// SIMATIC STEP 7 (V5.x) project EuroAsiaFood_V00_00_01
// CPU: CPU 314C-2 PN/DP
// station: Hardware
// station: SIMATIC 300(1)
// station: P_ADR_BUS
// program: S7-Programm(1)

SYMBOL_TABLE
"DB1 Weight Logging"	DB 1	FB 1	// Wiegemitschreibung
"DB2 Simulation"	DB 2	FB 2	// Simulation der Anlage
"DB3 global Info"	DB 3	DB 3	// globale Programm- / Fehlerinformationen
"DB4 Motor Data for FCs"	DB 4	DB 4	// Motordaten für Frequenzumformer
"DB5 reserve"	DB 5	DB 5	// reserve
"DB6 reserve"	DB 6	DB 6	// reserve
"DB7 SiSc-Par WS-Communic"	DB 7	DB 7	// Lagerort-Waagenparameter für WS Kopplung
"DB8 Batch Info from PC"	DB 8	DB 8	// Chargeninfo von PC
"DB9 reserve"	DB 9	DB 9
"DB10 Scale Configuration"	DB 10	DB 10	// Waagenkonfiguration
"DB11 Com DB Recipe Data"	DB 11	DB 11	// Koppel-DB Rezeptdaten
"DB12 Com-DB S-S Param"	DB 12	DB 12	// Koppel-DB Silo-Waagen-Parameter
"DB13 Scale Par from PC"	DB 13	DB 13	// SST Waagenparameter von PC
"DB14 Scale Par to PC"	DB 14	DB 14	// SST Waagenparameter zu PC
"DB15 R->C Level scale(S)"	DB 15	DB 15	// SST Rezeptebene -> Komponentenebene Waage Steuer-/Status
"DB16 R->C Level(D)"	DB 16	DB 16	// Interface recipe level  -> component level scale Data
"DB17 C->R Level Scale"	DB 17	DB 17	// SST Komponentneebene -> Rezeptebene Waage
"DB18 R<->C-Level Scale(A"	DB 18	DB 18	// SST Komponentneebene <-> Rezeptebene Waage Zusatzdaten
"DB19 DB Act Scale Data"	DB 19	DB 19	// Waagenistdaten-DB
"DB20 IF SC1 Control-DB"	DB 20	FB 15	// SST FG 1 <-> SPS-Waage Steuer-DB
"DB21 IF SC1 Scale Par"	DB 21	DB 21	// SST FG 1 <-> SPS-Waage Waagenparameter
"DB22 IF SC1 Recipe Data"	DB 22	DB 22	// SST FG 1 <-> SPS-Waage Lagerort-/Rezeptdaten
"DB23 IF SC2 Control-DB"	DB 23	FB 15	// SST FG 2 <-> SPS-Waage Steuer-DB
"DB24 IF SC2 Scale Par"	DB 24	DB 24	// SST FG 2 <-> SPS-Waage Waagenparameter
"DB25 IF SC2 Recipe Data"	DB 25	DB 25	// SST FG 2 <-> SPS-Waage Lagerort-/Rezeptdaten
"DB26 IF SC3 Control-DB"	DB 26	FB 15	// SST FG 3 <-> SPS-Waage Steuer-DB
"DB27 IF SC3 Scalen Par"	DB 27	DB 27	// SST FG 3 <-> SPS-Waage Waagenparameter
"DB28 IF SC3 Recipe Data"	DB 28	DB 28	// SST FG 3 <-> SPS-Waage Lagerort-/Rezeptdaten
"DB29 reserve"	DB 29	DB 29	// reserve
"DB30 Daten from/to SCADA"	DB 30	FB 30
"DB31 Mode to SCADA"	DB 31	DB 31	// Betriebsmode der Objekte zu Farbgrafik
"DB32 Inputs"	DB 32	FB 32
"DV33 Outputs"	DB 33	FB 33
"DB34 Faults"	DB 34	FB 34	// Anlagenstörungen
"DB35 Acknowledge Faults"	DB 35	DB 35	// Quittierungen
"DB36 Operating notific"	DB 36	DB 36	// Betriebsmeldungen
"DB37Service warning msg"	DB 37	DB 37	// Service Warnmeldungen
"DB38 Service fault msg"	DB 38	DB 38	// Service Störmeldungen
"DB39 free Data for SCADA"	DB 39	DB 39	// freie Datenaufzeichnung über Visualisierung
"DB40 IF SC4 Control-DB"	DB 40	FB 15	// SST FG 4 <-> SPS-Waage Steuer-DB
"DB41 IF SC4 Scale Par"	DB 41	DB 41	// SST FG 4 <-> SPS-Waage Waagenparameter
"DB42 IF SC4 Recipe Data"	DB 42	DB 42	// SST FG 4 <-> SPS-Waage Lagerort-/Rezeptdaten
"DB43 IF SC5 Control-DB"	DB 43	FB 15	// SST FG 5 <-> SPS-Waage Steuer-DB
"DB44 IF SC5 Scale Par"	DB 44	DB 44	// SST FG 5 <-> SPS-Waage Waagenparameter
"DB45 IF SC5 Recipe Data"	DB 45	DB 45	// SST FG 5 <-> SPS-Waage Lagerort-/Rezeptdaten
"DB46 IF SC6 Control-DB"	DB 46	FB 15	// SST FG 6 <-> SPS-Waage Steuer-DB
"DB47 IF SC6 Scale Par"	DB 47	DB 47	// SST FG 6 <-> SPS-Waage Waagenparameter
"DB48 IF SC6 Recipe Data"	DB 48	DB 48	// SST FG 6 <-> SPS-Waage Lagerort-/Rezeptdaten
"DB49 reserve"	DB 49	DB 49	// reserve
"DB50 Control bits PC"	DB 50	DB 50	// Steuerbitleiste von/zu PC
"DB51 Manual Addition PC"	DB 51	DB 51	// Quittierung Handzugaben / Daten Handzugaben von/zu PC
"DB52 Batch Info PC"	DB 52	DB 52	// Chargeninformationen von PC (Rezeptnr./Chargennr. usw.)
"DB53 Consumer Info PC"	DB 53	DB 53	// Verbraucherinformationen von/zu PC
"DB54 Transponder Info PC"	DB 54	DB 54	// Transponderinfprmationen von/zu PC
"DB55 Silo Info PC"	DB 55	DB 55	// Siloinformationen von/zu PC
"DB56 Silo Refill"	DB 56	DB 56	// Silonachfüllung von/zu PC
"DB57 List Man Addition"	DB 57	DB 57	// Handzugabeliste zur Anzeige auf OP oder FG)
"DB58 Project spec. res."	DB 58	DB 58	// reserve
"DB59 Mixer Values"	DB 59	DB 59	// Mischerwerte an PC
"DB60 Mixer Step Info"	DB 60	DB 60	// Mischerschrittinformationen an PC
"DB61 Mix Recipe M1"	DB 61	DB 61	// Mixer Recipe Mixerer 1 bzw. Heating Mixer 1 and Cooling Mixerer 1 from PC
"DB62 Mix Recipe M2"	DB 62	DB 62	// Mixer recipe mixer 2 or heater mixer 2 and cooler mixer 2 from PC
"DB63 Mix Recipe M3"	DB 63	DB 63	// Mixer recipe mixer 3 or heater mixer 3 and cooler mixer 3 from PC
"DB64 Mix Recipe M4"	DB 64	DB 64	// Mixer recipe mixer 4 or heater mixer 4 and cooler mixer 4 from PC
"DB65 Mix Recipe M5"	DB 65	DB 65	// Mixer recipe mixer 5 or heater mixer 5 and cooler mixer 5 from PC
"DB66 Mix Recipe M6"	DB 66	DB 66	// Mixer recipe mixer 6 or heater mixer 6 and cooler mixer 6 from PC
"DB67 Mix Recipe M7"	DB 67	DB 67	// Mixer recipe mixer 7 or heater mixer 7 and cooler mixer 7 from PC
"DB68 Mix Recipe M8"	DB 68	DB 68	// Mixer recipe mixer 8 or heater mixer 8 and cooler mixer 8 from PC
"DB69 Mix Recipe M9"	DB 69	DB 69	// Mixer recipe mixer 9 or heater mixer 9 and cooler mixer 9 from PC
"DB70 IF OP1 Control-DB"	DB 70	FB 16	// SST OP 1 <-> SPS-Waage Steuer-DB
"DB71 IF OP1 Scale Par"	DB 71	DB 71	// SST OP 1 <-> SPS-Waage Waagenparameter
"DB72 IF OP1 Recipe Datan"	DB 72	DB 72	// SST OP 1 <-> SPS-Waage Lagerort-/Rezeptdaten
"DB73 IF OP2 Control-DB"	DB 73	FB 16	// SST OP 2 <-> SPS-Waage Steuer-DB
"DB74 IF OP2 Scale Par"	DB 74	DB 74	// SST OP 2 <-> SPS-Waage Waagenparameter
"DB75 IF OP2 Recipe Data"	DB 75	DB 75	// SST OP 2 <-> SPS-Waage Lagerort-/Rezeptdaten
"DB90 Shuttle-DB"	DB 90	DB 90	// Shuttle-DB
"DB91 ContainerDB Shuttle"	DB 91	DB 91	// Container-DB Shuttle
"DB92 Station-DB Shuttle"	DB 92	DB 92	// Stations-DB Shuttle
"PRODUCTION_DB"	DB 1000	FB 1000	// Call Line 1 DB
"HOPPER_HP01_DB"	DB 1001	FB 1001
"HOPPER_HP02_DB"	DB 1002	FB 1001
"REC01_DB"	DB 1011	FB 1011	// Receiver REC01
"PMP01_DB"	DB 1051	FB 1051
"FC01_RV_HOPPERS_DB"	DB 10001	FB 4901
"Example DB read table"	DB 60000	DB 60000	// Beispiel-DB Tabelle auslesen
"R->C Level Scale (S)"	DB 60201	DB 60201	// SST Rezeptebene -> Komponentenebene Waage Steuer-/Status
"R->C Level Scale (D)"	DB 60202	DB 60202	// SST Rezeptebene -> Komponentenebene Waage Daten
"K->S Level Scale (S)"	DB 60203	DB 60203	// SST Komponentenebene -> Einzelschrittebene Waage Steuer-/Status
"K->S Level Scale (D)"	DB 60204	DB 60204	// Interface component level -> single step level Scale Daten
"S->A Level Scale (S)"	DB 60205	DB 60205	// SST Einzelschrittebene -> Analogebene Waage Steuer-/Status
"S->A Level Scale (D)"	DB 60206	DB 60206	// SST Einzelschrittebene -> Analogebene Waage Daten
"K->R Level Scale"	DB 60207	DB 60207	// SST Komponentneebene -> Rezeptebene Waage
"S->C Level Scale"	DB 60208	DB 60208	// SST Einzelschrittebene -> Komponentenebene Waage
"A->S Level Scale"	DB 60209	DB 60209	// SST Analogebene -> Einzelschrittebene Waage
"IF SCADA Control-DB"	DB 60211	DB 60211	// Schnittstelle zu Farbgrafik Steuer-DB
"IF SCADA Scale Par"	DB 60212	DB 60212	// Schnittstelle zu Farbgrafik Waagenparameter
"IF SCADA RecipeData"	DB 60213	DB 60213	// Schnittstelle zu Farbgrafik Rezeptdaten
"IF SCADA 1 Control-DB"	DB 60250	DB 60250	// SST FG 1 <-> SPS-Waage Steuer-DB
"Mixer Recipe-DB"	DB 60300	DB 60300	// Mixer recipe DB
"FB1 Weight logging"	FB 1	FB 1	// Wiegemitschreibung
"FB2 Simulation"	FB 2	FB 2	// Simulation der Anlage
"FB3 Mix Recipe Interpr."	FB 3	FB 3	// Mischrezeptinterpreter
"FB4 Freq Converter L2"	FB 4	FB 4	// Frequenzumformer L2-Bus
"FB5 Componenter_L2"	FB 5	FB 5	// Componenter L2-Bus
"FB6 reserve"	FB 6	FB 6	// reserve
"FB7 Rot Diverter Valve"	FB 7	FB 7	// Saugrohrverteiler
"FB8 reserve"	FB 8	FB 8	// reserve
"FB9 Pos. Pipe Diverter"	FB 9	FB 9	// Wegstellung (Rohrweiche)
"FB10 Order Level"	FB 10	FB 10	// Auftragsebene Waage
"FB11 Recipe Level"	FB 11	FB 11	// Rezeptebene Waage
"FB12 Component Level"	FB 12	FB 12	// Komponentenebene Waage
"FB13 Single Step Level"	FB 13	FB 13	// Single step level scale
"FB14 Analogue Level"	FB 14	FB 14	// Analogue level scale
"FB15 IF PLC-Scale/SCADA"	FB 15	FB 15	// Schnittstelle SPS-Waage / Farbgrafik
"FB16 IF PLC-Scale/OP"	FB 16	FB 16	// Schnittstelle SPS-Waage / OP
"FB17 IF PLC-Scale/HSH"	FB 17	FB 17	// Schnittstelle SPS-Waage / HSH
"FB18 IF PLC-Scale/OP OL"	FB 18	FB 18	// Schnittstelle SPS-Waage / OP Auftragebene
"FB19 IF PLC-Scale/Bil"	FB 19	FB 19	// Schnittstelle SPS-Waage / Farbgrafik Bilanzen
"FB20 Siwarex-U Comm"	FB 20	FB 20	// SPS-Waage Siwarex-U Kopplung
"FB21 MCS-DMV Comm"	FB 21	FB 21	// SPS-Waage MCS-DMV Kopplung
"FB22 MV1 Comm"	FB 22	FB 22	// SPS-Waage MV1 Kopplung
"FB23 Siwarex-M Comm"	FB 23	FB 23	// SPS-Waage Siwarex-M Kopplung
"FB25 Promass 63 Comm"	FB 25	FB 25	// SPS-Waage Promass 63 Kopplung
"FB26 Pulse Count FM350-2"	FB 26	FB 26	// SPS-Waage Impulszähler FM350-2 Kopplung
"FB27 PESA"	FB 27	FB 27	// SPS-Waage PESA Modul Kopplung
"FB28 Bizerba"	FB 28	FB 28	// SPS-Waage Bizerba Modul Kopplung
"FB29 Mettler-Scale ID7"	FB 29	FB 29	// SPS-Waage Mettler-ID7
"FB30 Daten from/to SCADA"	FB 30	FB 30	// Daten von / an Farbgrafik
"FB31 Mode Obj. to SCADA"	FB 31	FB 31	// Mode Objekte an Farbgrafik OP
"FB32 Inputs to SCADA"	FB 32	FB 32	// Eingänge an Farbgrafik / OP
"FB33 Outputs to SCADA"	FB 33	FB 33	// Ausgänge an Farbgrafik / OP
"FB34 Fault evaluation"	FB 34	FB 34	// Störauswertung
"FB36 WMD ET200M"	FB 36	FB 36	// SPS-Waage WMD Kopplung
"FB37 Pulse Count FM350-1"	FB 37	FB 37	// PLC-scale Pulse Counter FM 350-1
"FB38 gwt PR5210"	FB 38	FB 38	// SPS-Waage gwt PR5210
"FB39 WMD Bürkert"	FB 39	FB 39	// SPS-Waage WMD Bürkert
"FB40 Weight Siware- U"	FB 40	FB 40	// Gewichtswert von Siwarex U
"FB41 Weight MCS-DMV"	FB 41	FB 41	// Gewichtswert von MCS-DMV
"FB42 Weight MV1"	FB 42	FB 42	// Gewichtswert von MV1
"FB43 Weight Siwarex-M"	FB 43	FB 43	// Gewichtswert von Siwarex M
"FB45 LiW  DISOCONT"	FB 45	FB 45	// Differentialdosierwaage DSIOCONT
"FB46 IF LiW / SCADA"	FB 46	FB 46	// Schnittstelle DISOCONT Differentialdosierwaage / Farbgrafik
"FB47 IF LiW / OP"	FB 47	FB 47	// Schnittstelle DISOCONT Differentialdosierwaage / OP
"FB50 Control signals PC"	FB 50	FB 50	// Steuerbits von/an PC
"FB51 Manual addition"	FB 51	FB 51	// Quittierung Handzugaben / Daten Handzugabe
"FB52 Batch Info"	FB 52	FB 52	// Chargeninformationen (Rezept Nr./Chargennummer usw.)
"FB53 Consumer Info"	FB 53	FB 53	// Verbraucherinformationen von/zu PC
"FB54 Transponder Info"	FB 54	FB 54	// Transponderinformationen von/zu PC
"FB55 Silo Info PC"	FB 55	FB 55	// Siloinformationen von/zu PC
"FB56 Silo Refill"	FB 56	FB 56	// Silonachfüllung von/zu PC
"FB71 Siwarex CS"	FB 71	FB 71	// SPS-Waage Siwarex CS Kopplung Analogebene
"FB72 Siwarex CS_DR"	FB 72	FB 72	// SPS-Waage Siwarex CS Kopplung Siemens "SICS_DR"
"FB73 Siwarex CS_BA"	FB 73	FB 73	// SPS-Waage Siwarex CS Kopplung Siemens "SICS_BA"
"FB74 Counter ET200S"	FB 74	FB 74	// SPS-Waage Impulszähler über ET200S 1Count 24V/100kHz
"FB75 Mettler Jaguar"	FB 75	FB 75	// SPS-Waage Mettler Jaguar
"FB76 Siwarex FTA"	FB 76	FB 76	// SPS-Waage Siwarex FTA
"FB77 FB Siwarex FTA"	FB 77	FB 77	// SPS-Waage FB Siwarex FTA Siemens Funktionsbaustein
"FB78 Mettler PB-Module"	FB 78	FB 78	// SPS-Waage Mettler Profibus-Modul
"FB79 Mettler IND690"	FB 79	FB 79	// SPS-Waage Mettler IND690
"FB80 DK800"	FB 80	FB 80	// SPS-Waage DK800
"FB81 Promag 50"	FB 81	FB 81	// SPS-Waage Promag 50
"FB82 Mettler Panther"	FB 82	FB 82	// SPS-Waage Mettler Panther
"FB90 Shuttle-FB"	FB 90	FB 90	// Shuttle-FB
"FB91 ContainerFB Shuttle"	FB 91	FB 91	// Container-FB Shuttle
"FB92 Stations-FB Shuttle"	FB 92	FB 92	// Stations-FB Shuttle
"PRODUCTION"	FB 1000	FB 1000	// Call Line FBs
"HOPPER"	FB 1001	FB 1001	// HP01 and HP02
"REC01"	FB 1011	FB 1011	// Receiver REC01
"PMP01"	FB 1051	FB 1051
"BLOWER_P01"	FB 1081	FB 1081	// Pressure Blower
"FC01_RV_HOPPERS"	FB 4901	FB 4901	// Frequncy Converter rotary valves HP01/HP02
"FC1 Cycle Gen Timer"	FC 1	FC 1	// Taktgeber mit Timervorgabe
"FC2 Cycle Gen Timer Emul"	FC 2	FC 2	// Taktgeber mit Timernachbildung
"FC3 Cycle generator"	FC 3	FC 3	// Timernachbildung SA,SE,SV,SI
"FC4 Block transfer ANY"	FC 4	FC 4	// Block transferieren mit ANY-Zeiger
"FC5 Block Transfer"	FC 5	FC 5	// Block transferieren, Datenwort schreiben
"FC6 Set/Query Data Bit"	FC 6	FC 6	// Datenbit zuweisen oder abfragen
"FC7 Read Table"	FC 7	FC 7	// Eintrag aus Tabelle auslesen
"FC8 Determin ANY-Pointer"	FC 8	FC 8	// ANY-Zeiger in DB,DW,Länge zerlegen
"FC9 Set path"	FC 9	FC 9	// Weg stellen (Rohrweichen)
"FC10 Analogue value r/w"	FC 10	FC 10	// Analogwert lesen/schreiben
"FC11 PressureTransmitter"	FC 11	FC 11	// Drucktransmitterwert einlesen
"FC12 Restart"	FC 12	FC 12	// Neu- / Wiedeanlauf
"FC13 Standard Signals"	FC 13	FC 13	// Standardsignale
"FC14 Debounce Indicator"	FC 14	FC 14	// Melder entprellen
"FC15 I/O-FAT/Simulation"	FC 15	FC 15	// E/A FAT / Simulation
"FC16 Fault evaluation"	FC 16	FC 16	// Störauswertung
"FC17 String compare"	FC 17	FC 17	// Stringvergleich
"FC18 FIFO/LIFO"	FC 18	FC 18	// FIFO/LIFO
"FC19 Motor 2O2I"	FC 19	FC 19	// Motor Objekt 2 (2 Ausgänge, 2 Eingänge)
"FC20 Motor 1O1I"	FC 20	FC 20	// Motor Objekt 1 (1 Ausgang, 1 Eingang)
"FC21 Valve 10-2I"	FC 21	FC 21	// Ventil Objekt 1 (1 Ausgang, 0-2 Eingänge)
"FC22 Valve 2O2I"	FC 22	FC 22	// Ventil Objekt 2 (2 Ausgänge, 2Eingänge)
"FC23 Valve 1-10O"	FC 23	FC 23	// Ventil Objekt 3 (Ansteuerung von max. 10 getakteten Ventilen)
"FC24 Binary-I Object"	FC 24	FC 24	// Binär-Eingangs Objekt
"FC25 Pipe Diverter 3O3I"	FC 25	FC 25	// Pipe Diverter 3 Outputs, 3 inputs
"FC26 DosingValve 2O2I"	FC 26	FC 26	// Dosierventil grob/fein 2 Ausgänge, 2 Eingänge)
"FC30 Pre -assign DB"	FC 30	FC 30	// Datenbaustein vorbelegen
"FC31 PLC-Scale"	FC 31	FC 31	// Aufruf SPS-Waage
"FC32 Rec/Comp r/w/d"	FC 32	FC 32	// Rezept/Komponente lesen/schreiben/löschen
"FC33 Si/Rec from PC r/w"	FC 33	FC 33	// Lagerortparameter von PC lesen/schreiben
"FC34 Si/Sc Par r/w"	FC 34	FC 34	// Silo-/Waagenparameter lesen/schreiben
"FC35 reserve Scale"	FC 35	FC 35
"FC36 Si-Configuration"	FC 36	FC 36	// Lagerortkonfiguration
"FC37 Si/Sc Par r/w"	FC 37	FC 37	// Lagerortparameter einer Siwarex-Waage lesen/schreiben
"FC38 reserve Scale"	FC 38	FC 38
"FC39 Siwarex-M"	FC 39	FC 39	// Kommunikationsbaustein Siwarex-M
"FC40 copy Obj-IF Master"	FC 40	FC 40	// Objekt-Schnittstelle kopieren Master
"FC41 copy Obj-IF Slave"	FC 41	FC 41	// Objekt-Schnittstelle kopieren Slave
"FC43 FM350-2"	FC 43	FC 43
"FC44 FM350-2 I/O"	FC 44	FC 44
"FC45 Data Promass 63"	FC 45	FC 45	// Daten von Promass 63 DP
"FC47 Write Table"	FC 47	FC 47	// Eintrag in Tabelle schreiben
"FC50 LiW Scale DISOCONT"	FC 50	FC 50	// FC50 Aufruf DISOCONT Differentialdosierwaage
"FC60 Silo Pilot"	FC 60	FC 60	// Silopilot
"FC61 Bürkert DosingValve"	FC 61	FC 61	// Bürkert Dosierventil
"FC62 Analogue Valve"	FC 62	FC 62	// Analogventil
"FC64 aux fct registr"	FC 64	FC 64	// Hilfsfunktion Registrierung
"FC65 scale-db-no"	FC 65	FC 65
"FC66 info functiontime"	FC 66	FC 66
"EUi_02_04_201"	I 4.0	BOOL	// production area PMP01 motor vacuum pump
"EUi_02_01_201"	I 4.1	BOOL	// production area REC01 motor rotary valev
"EUi_02_02_201"	I 4.2	BOOL	// production area SM01 motor screener
"EUi_02_02_202"	I 4.3	BOOL	// production area SM01 motor magnetic seperator
"EUi_01_01_201"	I 4.4	BOOL	// material preparation HP01 motor rotary valve
"EUi_01_02_201"	I 4.5	BOOL	// material preparation HP02 motor rotary valve
"Ln_01_01_301"	I 4.6	BOOL	// material preparation HP01 low level sensor indicator
"Ln_01_02_301"	I 4.7	BOOL	// material preparation HP01 low level sensor indicator
"HZ_02_04_201"	I 5.0	BOOL	// production area PMP01 motor vacuum pump
"HZ_02_01_201"	I 5.1	BOOL	// production area REC01 motor rotary valve
"HZ_02_02_201"	I 5.2	BOOL	// production area SM01 motor screener
"HZ_02_02_202"	I 5.3	BOOL	// production area SM01 motor magnetic seperator
"HZ_01_01_201"	I 5.4	BOOL	// material preparation HP01 motor rotary valve
"HZ_01_02_201"	I 5.5	BOOL	// material preparation HP02 motor rotary valve
"ES_03_01_601"	I 5.6	BOOL	// system system input emergency stop ok
"ES_03_01_602"	I 5.7	BOOL	// system system input fault fuse
"GZ_02_01_601"	I 6.0	BOOL	// production area REC01 input safety circuit
"GZ_02_02_601"	I 6.1	BOOL	// production area SM01 input safety circuit
"GZ_01_01_601"	I 6.2	BOOL	// material preparation HP01 input safety circuit
"GZ_01_02_601"	I 6.3	BOOL	// material preparation HP02 input safety circuit
"Gn_02_01_602"	I 6.4	BOOL	// production area REC01 input rotor monitoring
"Gn_01_01_602"	I 6.5	BOOL	// material preparation HP01 input rotor monitoring
"Gn_01_02_602"	I 6.6	BOOL	// material preparation HP02 input rotor monitoring
"I 6.7"	I 6.7	BOOL	// free
"Lp_02_01_301"	I 10.0	BOOL	// production area REC01 sensor high level indicator
"Ln_02_01_302"	I 10.1	BOOL	// production area REC01 sensor low level indicator
"Lp_02_03_301"	I 10.2	BOOL	// production area HP03 sensor high level indicator
"Ln_02_03_302"	I 10.3	BOOL	// production area HP03 sensor low level indicator
"Gp_01_02_102"	I 10.4	BOOL	// material preparation HP02 valve outlet flap
"EUi_01_01_202"	I 10.5	BOOL	// material preparation HP01 motor vibrator
"EUi_01_02_202"	I 10.6	BOOL	// material preparation HP02 motor vibrator 1
"EUi_01_02_203"	I 10.7	BOOL	// material preparation HP02 motor vibrator 2
"HZ_01_01_202"	I 11.0	BOOL	// material preparation HP01 motor vibrator
"HZ_01_02_202"	I 11.1	BOOL	// material preparation HP02 motor vibrator 1
"HZ_01_02_203"	I 11.2	BOOL	// material preparation HP02 motor vibrator 2
"ES_02_03_601"	I 11.3	BOOL	// production area HP03 input PFC ready
"ES_02_03_602"	I 11.4	BOOL	// production area HP03 input PFC take material
"ES_01_02_603"	I 11.5	BOOL	// production area HP03 input PFC n.a
"ES_01_02_604"	I 11.6	BOOL	// production area HP03 input PFC n.a
"I 11.7"	I 11.7	BOOL	// free
"M 0.0 Lock Man.Operation"	M 0.0	BOOL	// Handbedienung zentral sperren
"M 0.1 Constant 1"	M 0.1	BOOL	// Merker konstant 1
"M 0.2 Constant 0"	M 0.2	BOOL	// Merker konstant 0
"M 0.3 Reset"	M 0.3	BOOL	// allgemeiner Reset
"M 0.4 reserve"	M 0.4	BOOL
"M 0.5 InternalSimulation"	M 0.5	BOOL	// Simulation intern ein
"M 0.6 Simulation AVP"	M 0.6	BOOL	// Simulation über AVP
"M 0.7 Battery empty"	M 0.7	BOOL	// Batterie leer
"M 1.0 Ack. faults"	M 1.0	BOOL	// Quittierung Störung
"M 1.1 general Fault"	M 1.1	BOOL	// allgemeine Stoerung
"M 1.2 First-out Fault"	M 1.2	BOOL	// Erstmeldung allgemeine Störung
"M 1.3 Hot/WarmRestartPLC"	M 1.3	BOOL	// Neustart oder Wiederanlauf SPS
"M 1.4 Cold Restart PLC"	M 1.4	BOOL	// Kaltstart PLC
"M 1.5 I/O FAT"	M 1.5	BOOL	// E/A FAT mit AVP
"M 1.6 ClckDdebounceIndic"	M 1.6	BOOL	// Takt Entprellung Füllstandsmelder
"M 1.7 Cycle Timer-FC"	M 1.7	BOOL	// Takt Timer-FC
"M 2.0 Cycle 0,1-sec"	M 2.0	BOOL	// Merker Takt 0,1 sek
"M 2.1 Cycle 0,2-sec"	M 2.1	BOOL	// Merker Takt 0,2 sek
"M 2.2 Cycle 0,4-sec"	M 2.2	BOOL	// Merker Takt 0,4 sek
"M 2.3 Cycle 0,5-sec"	M 2.3	BOOL	// Merker Takt 0,5 sek
"M 2.4 Cycle 0,8-sec"	M 2.4	BOOL	// Merker Takt 0,8 sek
"M 2.5 Cycle 1,0-sec"	M 2.5	BOOL	// Merker Takt 1,0 sek
"M 2.6 Cycle 1,6-sec"	M 2.6	BOOL	// Merker Takt 1,6 sek
"M 2.7 Cycle 2,0-sec"	M 2.7	BOOL	// Merker Takt 2,0 sek
"M 3.0 Flk Cycle 0,1-sec"	M 3.0	BOOL	// Flankenmerker Takt 0,1 sek
"M 3.1 Flk Cycle 0,2-sec"	M 3.1	BOOL	// Flankenmerker Takt 0,2 sek
"M 3.2 Flk Cycle 0,4-sec"	M 3.2	BOOL	// Flankenmerker Takt 0,4 sek
"M 3.3 Flk Cycle 0,5-sec"	M 3.3	BOOL	// Flankenmerker Takt 0,5 sek
"M 3.4 Flk Cycle 0,8-sec"	M 3.4	BOOL	// Flankenmerker Takt 0,8 sek
"M 3.5 Flk Cycle 1,0-sec"	M 3.5	BOOL	// Flankenmerker Takt 1,0 sek
"M 3.6 Flk Cycle 1,6-sec"	M 3.6	BOOL	// Flankenmerker Cycle 1,6 sek
"M 3.7 Flk Cycle 2,0-sec"	M 3.7	BOOL	// Flankenmerker Cycle 2,0 sek
"M 4.0 Imp Cycle 0,1-sec"	M 4.0	BOOL	// Impulsmerker Takt 0,1 sek
"M 4.1 Imp Cycle 0,2-sec"	M 4.1	BOOL	// Impulsmerker Takt 0,2 sek
"M 4.2 Imp Cycle 0,4-sec"	M 4.2	BOOL	// Impulsmerker Takt 0,4 sek
"M 4.3 Imp Cycle 0,5-sec"	M 4.3	BOOL	// Impulsmerker Takt 0,5 sek
"M 4.4 Imp Cycle 0,8-sec"	M 4.4	BOOL	// Impulsmerker Takt 0,8 sek
"M 4.5 Imp Cycle 1,0-sec"	M 4.5	BOOL	// Impulsmerker Takt 1,0 sek
"M 4.6 Imp Cycle 1,6-sec"	M 4.6	BOOL	// Impulsmerker Takt 1,6 sek
"M 4.7 Imp Cycle 2,0-sec"	M 4.7	BOOL	// Impulsmerker Takt 2,0 sek
"M 8.0 First-out alarm PC"	M 8.0	BOOL	// Erstmeldung an PC
"M 8.1 ACK Fault from PC"	M 8.1	BOOL	// Quittierung Störung von PC
"Service mode lock auto"	M 9.5	BOOL
"Lamp Testing"	M 9.7	BOOL	// flag to test all lamps of the system
"M 10.0 Motor ManOp rel"	M 10.0	BOOL	// Motor Handbedienung erlaubt
"M 10.1 Motor ACK nescess"	M 10.1	BOOL	// Motor Quittierung Störung nötig
"M 11.0 Valve ManOp rel"	M 11.0	BOOL	// Ventil Handbedienung erlaubt
"M 11.1 Valve ACK nescess"	M 11.1	BOOL	// Ventil Quittierung Störung nötig
"MB 2 Cycle Flags"	MB 2	BYTE	// Taktmerker (von CPU Hardwarekonfiguration)
"MB 3 Edge Flags MB2"	MB 3	BYTE	// Flankenmerker von Takten MB2
"MB 4 Pulse Flags MB2"	MB 4	BYTE	// Impulsmerker von Takten MB2
"MW 6 Timer Val Cycle FCs"	MW 6	INT	// Zeitwert Takt-FCs in 0,1s
"OB1 Cycle"	OB 1	OB 1	// Main Cycle
"OB 80 Zeitfehler-OB"	OB 80	OB 80	// Zeitfehler-OB
"OB 81 Stromversorg-OB"	OB 81	OB 81	// Stromversorgungsfehler-OB
"OB 82 Diagnosealarm-OB"	OB 82	OB 82	// Diagnosealamrn-OB
"OB 83 Ziehen-/Stecken-OB"	OB 83	OB 83	// Ziehen-/Stecke-OB
"OB 84 CPU-Hardwaref-OB"	OB 84	OB 84	// CPU-Hardwarefehler-OB
"OB 85 Prgablauffehler-OB"	OB 85	OB 85	// Programmablauffehler-OB
"OB 86 Baugr träger-OB"	OB 86	OB 86	// Baugruppenträgerausfall-OB
"OB 87 Kommunikations-OB"	OB 87	OB 87	// Kommunikationsfehler-OB
"OB 88 BREAKUP ERROR OB"	OB 88	OB 88	// Abortion of Processing
"OB 100 Neustart-OB"	OB 100	OB 100	// Neustart-OB
"OB 101 Wiederanlauf-OB"	OB 101	OB 101	// Wiederanlauf-OB
"OB 102 Kaltstart"	OB 102	OB 102	// Cold Restart
"OB 121 Programmierf-OB"	OB 121	OB 121	// Programmierfehler-OB
"OB 122 Peripheriezugr-OB"	OB 122	OB 122	// Peripheriezugriffsfehler
"EUq_02_04_201"	Q 4.0	BOOL	// production area PMP01 motor vacuum pump
"EUq_02_01_201"	Q 4.1	BOOL	// production area REC01 motor rotary valve
"EUq_02_02_201"	Q 4.2	BOOL	// production area SM01 motor screener
"EUq_02_02_202"	Q 4.3	BOOL	// production area SM01 motor magnetic seperator
"EUq_01_01_201"	Q 4.4	BOOL	// material preparation HP01 motor rotary valve
"EUq_01_02_201"	Q 4.5	BOOL	// material preparation HP02 motor rotary valve
"O 4.6"	Q 4.6	BOOL	// free
"O 4.7"	Q 4.7	BOOL	// free
"UVp_02_01_101"	Q 5.0	BOOL	// production area REC01 valve air purged bearing
"UVp_01_01_101"	Q 5.1	BOOL	// material preparation HP01 valve air purged bearing
"UVp_01_02_101"	Q 5.2	BOOL	// material preparation HP02 valve air purged bearing
"O 5.3"	Q 5.3	BOOL	// free
"O 5.4"	Q 5.4	BOOL	// free
"O 5.5"	Q 5.5	BOOL	// free
"O 5.6"	Q 5.6	BOOL	// free
"O 5.7"	Q 5.7	BOOL	// free
"UVp_02_01_102"	Q 10.0	BOOL	// production area REC01 valve air purged filter
"UVp_02_01_103"	Q 10.1	BOOL	// production area REC01 valve air purged filter
"UVp_02_01_104"	Q 10.2	BOOL	// production area REC01 valve air purged filter
"O 10.3"	Q 10.3	BOOL	// free
"O 10.4"	Q 10.4	BOOL	// free
"EUq_01_01_202"	Q 10.5	BOOL	// material preparation HP01 motor vibrator
"EUq_01_02_202"	Q 10.6	BOOL	// material preparation HP02 motor vibrator 1
"EUq_01_02_203"	Q 10.7	BOOL	// material preparation HP02 motor vibrator 2
"ES_02_01_501"	Q 11.0	BOOL	// production area HP01 output PFC
"ES_02_01_502"	Q 11.1	BOOL	// production area HP01 output PFC
"O 11.2"	Q 11.2	BOOL	// free
"ES_02_03_501"	Q 11.3	BOOL	// production area HP03 output PFC Product HP03
"ES_02_03_502"	Q 11.4	BOOL	// production area HP03 output PFC active
"ES_02_03_503"	Q 11.5	BOOL	// production area HP02 output PFC
"ES_02_03_504"	Q 11.6	BOOL	// free
"ES_02_03_505"	Q 11.7	BOOL	// collective fault
"SFB 12 BSEND"	SFB 12	SFB 12	// Block Oriented Send
"SFB 13 BRCV"	SFB 13	SFB 13	// Block Oriented Receive
"SET_CLK"	SFC 0	SFC 0	// Set System Clock
"READ_CLK"	SFC 1	SFC 1	// Read System Clock
"SFC 13 DPNRM_DG"	SFC 13	SFC 13	// Read Diagnostic Data of a DP Slave
"SFC 14 DPRD_DAT"	SFC 14	SFC 14	// Read DP Slave Record
"SFC 15 DPWR_DAT"	SFC 15	SFC 15	// Write DP Slave Record
"SFC 20 BLKMOV"	SFC 20	SFC 20	// Direct Word Move
"SFC 24 TEST_DB"	SFC 24	SFC 24	// Test Data Block
"RDSYSST"	SFC 51	SFC 51	// Read a System Status List or Partial List
"DatumUhrzeit"	VAT 1	
"_IO_ALL"	VAT 2	
"___IO_MotorsValves"	VAT 13	
"____IO_Allgemein"	VAT 31	
END_SYMBOL_TABLE

FUNCTION_BLOCK "FB2 Simulation"	// FB 2
TITLE = Simulation
//Creation:
//Date:            Author:                                               Version
//--------------------------------------------------------------------------------
//12.05.2016      Huang Qinsong (hqs)                                    01.00.00
//
//Changes:
//No. Date:        Who       Description                           Mark   Version 
//--------------------------------------------------------------------------------
//01
//________________________________________________________________________________
//Function:
//
VERSION : 0.1
VAR
  REC01 : STRUCT
   Weight : REAL ;
   SpeedFilling : REAL ;
   SpeedDischarging : REAL ;
  END_STRUCT ;
  HP03 : STRUCT
   Weight : REAL ;
   SpeedFilling : REAL ;
   SpeedDischarging : REAL ;
  END_STRUCT ;
END_VAR
BEGIN
NETWORK
TITLE = simulation condition
      AN    "M 0.5 InternalSimulation";
      BEC;
NETWORK
TITLE = PFKs
      SET;
      =     "ES_02_03_602";
NETWORK
TITLE =
      SET;
      =     "Gp_01_02_102";
NETWORK
TITLE = --- level indicator, HZ, GZ ---
      O     "M 1.3 Hot/WarmRestartPLC";
      O     "M 1.4 Cold Restart PLC";
      JCN   m001;
//system 
      S     "ES_03_01_601";
      S     "ES_03_01_602";
//REC01 01
//      S     "Lp_02_01_301"
//      S     "Ln_02_01_302"
// HP03
//      S     "Lp_02_03_301"
//     S     "Ln_02_03_302"
// Safety
      S     "GZ_02_01_601";
      S     "GZ_02_02_601";
      S     "GZ_01_02_601";
      S     "Gn_02_01_602";
      S     "Gn_01_01_602";
      S     "Gn_01_02_602";
//repair switches 
      S     "HZ_02_01_201";
      S     "HZ_02_04_201";
      S     "HZ_02_02_201";
      S     "HZ_02_02_202";
      S     "HZ_01_01_201";
      S     "HZ_01_02_201";
      S     "HZ_01_01_202";
      S     "HZ_01_02_202";
      S     "HZ_01_02_203";
NETWORK
TITLE = --- motors ---
      A     "EUq_02_04_201";
      =     "EUi_02_04_201";
      A     "EUq_02_01_201";
      =     "EUi_02_01_201";
      A     "EUq_02_02_201";
      =     "EUi_02_02_201";
      A     "EUq_02_02_202";
      =     "EUi_02_02_202";
      A     "EUq_01_01_201";
      =     "EUi_01_01_201";
      A     "EUq_01_02_201";
      =     "EUi_01_02_201";
      A     "EUq_01_02_202";
      =     "EUi_01_02_202";
      A     "EUq_01_02_203";
      =     "EUi_01_02_203";
      A     "EUq_01_01_202";
      =     "EUi_01_01_202";
NETWORK
TITLE = REC01 simulation
// SPEEDS DEFINITIONS
//   L     0.000000e+000
//      T     #REC01.Weight
// Speed Filling from HP01/HP02
      L     1.000000e+00;
      L     DB10001.DBD 58;
      *R;
      L     2.000000e+01;
      /R;
      T     #REC01.SpeedFilling;
// Speed Discharging 
      L     1.200000e+00;
      T     #REC01.SpeedDischarging;
// Filling
      A(;
      O     "EUi_01_01_201";
      O     "EUi_01_02_201";
      );
      A     "EUi_02_04_201";
      A     "M 4.5 Imp Cycle 1,0-sec";
      JCN   NFA;	//no production active
      L     #REC01.Weight;
      L     #REC01.SpeedFilling;
      +R;
      T     #REC01.Weight;
NFA:  NOP   0;
// Discharging 
      A     "EUi_02_01_201";
      A(;
      L     #REC01.Weight;
      L     0.000000e+00;
      >R;
      );
      A     "M 4.5 Imp Cycle 1,0-sec";
      JCN   NDA;	//no production active
      L     #REC01.Weight;
      L     #REC01.SpeedDischarging;
      -R;
      T     #REC01.Weight;
NDA:  NOP   0;
// low Level indicator
      A(;
      L     #REC01.Weight;
      L     2.000000e+01;
      >R;
      );
      NOT;
      =     "Ln_02_01_302";
// high Level Indicator
      A(;
      L     #REC01.Weight;
      L     1.000000e+02;
      >R;
      );
      NOT;
      =     "Lp_02_01_301";
NETWORK
TITLE = HP03 simulation
// SPEEDS DEFINITIONS
      L     #REC01.SpeedDischarging;
      T     #HP03.SpeedFilling;	//AZO Speed 
      L     1.000000e+00;
      T     #HP03.SpeedDischarging;	// Rovema Speed
// Filling
      A     "EUi_02_02_202";
      A     "M 4.5 Imp Cycle 1,0-sec";
      JCN   NDH;	//no production active
      L     #HP03.Weight;
      L     #HP03.SpeedFilling;
      +R;
      T     #HP03.Weight;
NDH:  NOP   0;
//Discharging
      A     "ES_02_03_602";
      A     "M 4.5 Imp Cycle 1,0-sec";
      A(;
      L     #HP03.Weight;
      L     0.000000e+00;
      >R;
      );
      JCN   NDD;
      L     #HP03.Weight;
      L     #HP03.SpeedDischarging;
      -R;
      T     #HP03.Weight;
NDD:  NOP   0;
      A(;
      L     #HP03.Weight;
      L     1.000000e+01;
      >R;
      );
      NOT;
      =     "Ln_02_03_302";
      A(;
      L     #HP03.Weight;
      L     1.000000e+02;
      >R;
      );
      NOT;
      =     "Lp_02_03_301";
NETWORK
TITLE =
// =================================================
      SET;
//      =     "Ln_01_01_301"
//     =     "Ln_01_02_301"
      SET;
      =     "HZ_02_04_201";
      =     "HZ_02_01_201";
      =     "HZ_02_02_201";
      =     "HZ_02_02_202";
      =     "HZ_01_01_201";
      =     "HZ_01_02_201";
      SET;
      =     "GZ_02_01_601";
      =     "GZ_02_02_601";
      =     "GZ_01_01_601";
      =     "GZ_01_02_601";
      SET;
      =     "Gn_02_01_602";
      =     "Gn_01_01_602";
      =     "Gn_01_02_602";
      SET;
//   =     "Lp_02_01_301"
//    =     "Ln_02_01_302"
//      =     "Lp_02_03_301"
//      =     "Ln_02_03_302"
      SET;
      =     "HZ_01_01_202";
      =     "HZ_01_02_202";
      =     "HZ_01_02_203";
      A     "EUq_02_04_201";
      =     "EUi_02_04_201";
      A     "EUq_02_02_202";
      =     "EUi_02_02_202";
// =================================================
NETWORK
TITLE = END
m001: NOP   0;
      SET;
      =     "ES_02_03_601";
      =     "ES_02_03_602";
      SET;
      =     "Lp_02_01_301";
      SET;
      =     "Ln_02_01_302";
      SET;
      =     "Lp_02_03_301";
      SET;
      =     "Ln_02_03_302";
      SET;
      =     "Ln_01_01_301";
      =     "Ln_01_02_301";
END_FUNCTION_BLOCK

FUNCTION_BLOCK "FB4 Freq Converter L2"	// FB 4
TITLE = Steuerung von SEW-Frequenzumf. mit DFP21B über Profibus-DP
//Building:
//Date         Editor                                                     Version
//--------------------------------------------------------------------------------
//11.12.06     R.Schaffert (sra)                                          01.00.00
//
//Modifications:
//No. Date     Edit  Description                                    Index Version
//--------------------------------------------------------------------------------
//01  12.04.07 sra   Ausgangsstrom in Ampere ausgeben               (001) 01.00.01
//02  23.06.10 sra   Betriebsmeldung mit Komm.fehlern erweitert     (002) 01.00.02
//03  19.10.11 sra   Begrenzung maximale Solldrehzahl               (003) 01.01.00
//04  19.03.12 sra   Änderung wegen Firmwareänderung SEW            (004) 01.01.01
//05  23.07.14 sra   Umschaltung Parametersatz eingefügt            (005) 01.02.00
//05  23.09.14 sra   Fehlerbeseitigung "Warnung"                    (006) 01.02.01
//06  23.11.15 kst   Fehlerbeseitigung allgemein                    (007) 01.03.00
//07  17.02.16 sra   out_FB_Fehlermeldung = INT                     (008) 01.03.01
//________________________________________________________________________________
//Functional description:
//
//The block communicates with SEW frequency converters MOVITRAC B via 
//Profibus interface DFP21B.
//
//Note:
//With this frequency converter it is not possible to transfer motor data.
//To be sure that the output value of the current is correct, the paramter 
//nominal motor current at the frequency convetrer must be set to correct value.
//
//Hardware configuration:
//
//Install GSD file in hardware catalogue:
// SEW_6009.GSD (Internet: www.SEW-EURODRIVE.de)
//
//The "Gateway DFP/DFS" Profibus module is then in the hardware catalogue under 
//the menu: "other field devices->Drives->SEW->DPV1->"
//Add this module to hardware and configure following modules
//     Slot 1: Empty
//     Slot 2: Parameter channel (8 byte)  with I/O address Z
//from Slot 3: AS Y Drives (Y x 3PD)       with I/O address Z+8 and following
//             where Y = Number of FCs 
//
//
//!!! The nominal motor frequency, motor speed and the nominal motor current must 
//    be transferred to ensure the block functions correctly.
//
//Settings at DFP21B:
//
//1. Set Profibus address via DIP switches on DFP21B: 
//
//2. Execute auto setup at DFP21B by setting DIP switch 8 (AS) to ON
//   All FCs must be switched on and the SBus address set
//   With the auto setup function (DIP switch "AS") it is possible to set up 
//   DFP21B as the gateway without a PC. The function is executed once when the 
//   DIP switch is switched on. The DIP switch must then remain on. The function 
//   can be executed again by switching the DIP switch off and on again.
//
//
//Frequency converter settings
//
//1. P100 Set setpoint source to SBUS -> value = 10
//
//2. P101 Set control source to SBus -> value 3
//
//3. P301 Set minimum speed in rpm (master value = 15)
//
//4. P302 Set maximum speed in rpm (factory setting = 1500)
//
//5. P303 Set current limit (in % of FC nominal current)
//   (Factory setting =150%)
//
//6. P320 Set automatic motor matching to on (standard setting)
//   (to gauge the motor at start)
//
//7. P500 Switch on speed monitoring
//   (in the case of fault messages P501 increase speed monitoring delay time)
//
//8. P601, P603 and P608 Set binary inputs to ""no function" (=0)
//   Set P602 to 1 = enable (factory setting) DI03 must be bypassed
//
//9. P604 for operation with PTC resistor set to 26 (TF message) otherwise
//.... zeroing.
//   
//11. P881 Set SBus address of respective frequency converter (from 1 in
//    ascending order)
//
//12. P883 Bus monitoring time -> 5 [s]
//
//13. P884 Check SBus baud rate -> value 500/500 kBaud
//
//14. P870-P872 Setpoint description PA1-PA3
//       P870 = control word 1
//       P871 = speed
//       P872 = reserve
//    P873-P876 Actual value description PE1-PE3
//       P873 = status word 1
//       P874 = speed
//       P875 = output current in % of nominal current
//
//Notice to Index/Modification (004):
//The firmware has been changed because some faults must be resetet with an 
//internal function and some other with an acknowledge function. If there has 
//been 
//an fault of the Thermocontact is wasn't necessary to reset the fault and the 
//frequency converter still signals "ready for operation". This also happened 
//with other fault messages. For the Profibus communication it wasn't possible to 
//detect what happend with the motor. Finally the function always signals always 
//a fault message.
//
AUTHOR : sra
FAMILY : AZO
VERSION : 0.0
VAR_INPUT
  in_PEA_Adresse : INT ;	//Basisadresse für EA-Daten im PEA-Bereich
  in_FU_Nummer : INT ;	//FU Nummer zur Berechnung des Offsets der Peripherie-EAs
  in_Auswahl_Param_satz_2 : BOOL ;	//Motorparametersatz 2 wird ausgewählt (bei Ansteuerung von 2 versch. Motortypen)
  in_Freigabe : BOOL ;	//Steuersignal 1 setzen zum Starten des FUs
  in_Linkslauf : BOOL ;	//Frequenzumformer Linkslauf ein
  in_Quittierung_Stoerung : BOOL ;	//Störung quittieren
  in_Sollfrequenz : REAL ;	//Sollfrequenz in Hz
  in_Motorleistungsfaktor : REAL ;	//nicht vorhanden => 0
  in_Motornennfrequenz : REAL ;	//Wertebereich: 0 - 100 Hz
  in_Motornenndrehzahl : REAL ;	//Wertebereich: 0 - 10000 U/min
  in_Motornennstrom : REAL ;	//Wertebereich: 0- ... A !! Hier muss der Stromwert des FUs eingegeben werden !!
  in_Motornennspannung : REAL ;	//nicht vorhanden => 0
  in_Motornennleistung : REAL ;	//nicht vorhanden => 0
END_VAR
VAR_OUTPUT
  out_Istfrequenz : REAL ;	//Istfrequenz in Hz
  out_Istdrehzahl : REAL ;	//Istdrehzahl in U/min
  out_Leistung : REAL ;	//nicht vorhanden => 0
  out_Drehmoment : REAL ;	//nicht vorhanden => 0
  out_Motorspannung : REAL ;	//nicht vorhanden => 0
  out_Ausgangsstrom : REAL ;	//Ausgangsstrom des FU
  out_Stoerung : BOOL ;	//1=Gerätestörung
  out_Warnung : BOOL ;	//1=max. Solldrehzahl überschritten
  out_Sollwert_erreicht : BOOL ;	//zeigt 1 an, wenn Istwert gleich Sollwert ist
  out_laeuft : BOOL ;	//=1 wenn Istdrehzahl > 0
  out_FB_Fehlermeldung : INT ;	//0 = ok ; sonst Fehler_Code_L2Dp (008)
  out_Stoerungsnummer : DINT ;	//Stoerungsnummer, bzw. Betriebszustand wenn keine Störung aktiv
END_VAR
VAR
  reserve : ARRAY  [58 .. 99 ] OF BYTE ;
  Parameterkanal_in : STRUCT
   Verwaltung_Subindex : STRUCT
    Dienst_Kennung_0 : BOOL ;
    Dienst_Kennung_1 : BOOL ;
    Dienst_Kennung_2 : BOOL ;
    Dienst_Kennung_3 : BOOL ;
    Datenlaenge_0 : BOOL ;
    Datenlaenge_1 : BOOL ;
    Handshake : BOOL ;
    Status_Bit : BOOL ;
    Subindex : BYTE ;
   END_STRUCT ;
   Parameter_Index : WORD ;
   Daten_1_2 : INT ;
   Daten_3_4 : INT ;
  END_STRUCT ;
  Parameterkanal_out : STRUCT
   Verwaltung_Subindex : STRUCT
    Dienst_Kennung_0 : BOOL ;
    Dienst_Kennung_1 : BOOL ;
    Dienst_Kennung_2 : BOOL ;
    Dienst_Kennung_3 : BOOL ;
    Datenlaenge_0 : BOOL ;
    Datenlaenge_1 : BOOL ;
    Handshake : BOOL ;
    Status_Bit : BOOL ;
    Subindex : BYTE ;
   END_STRUCT ;
   Parameter_Index : WORD ;
   Daten_1_2 : INT ;
   Daten_3_4 : INT ;
  END_STRUCT ;
  Prozessdatenkanal_in : STRUCT 	//Prozesseingangsdaten
   PI1_Statuswort : STRUCT
    Zustand_Fehlercode : BYTE ;
    Endstufe_freigegeben : BOOL ;
    Umrichter_betriebsbereit : BOOL ;
    PA_Daten_freigegeben : BOOL ;
    reserve_3 : BOOL ;
    akt_Parametersatz_2 : BOOL ;	//0 = 1. Satz; 1 = 2. Satz
    Stoerung_Warnung : BOOL ;
    reserve_6 : BOOL ;	//
    reserve_7 : BOOL ;	//
   END_STRUCT ;
   PI2_Istdrehzahl : INT ;
   PI3_Ausgangsstrom : INT ;
  END_STRUCT ;
  Prozessdatenkanal_out : STRUCT 	//Prozessausgangsdaten
   PO1_Steuerwort : STRUCT
    Drehrichtung : BOOL ;	//0 = rechts; 1 = links
    Motorpoti_auf : BOOL ;	//00=11= keine Änderung; 01=Hochlauf, 02=Tieflauf
    Motorpoti_ab : BOOL ;
    Festsollwerte_0 : BOOL ;	//00 = Feldbus
    Festsollwerte_1 : BOOL ;
    Festsollwert_Umschaltung : BOOL ;
    reserve_14 : BOOL ;
    reserve_15 : BOOL ;
    Reglersperre : BOOL ;	//Freigabe = '110', sonst Halt
    Freigabe_Schnellstop : BOOL ;
    Freigabe_Normalhalt : BOOL ;
    reserve_3 : BOOL ;
    Integratorauswahl : BOOL ;	//0 = Integrator 2; 1 = Integrator 1 (005) noch nicht verwendet
    Parametersatz_2 : BOOL ;	//0 = Parametersatz 1; 1 = Parametersatz 2 (005)
    Reset_Stoerung : BOOL ;	//
    reserve_7 : BOOL ;
   END_STRUCT ;
   PO2_Solldrehzahl : INT ;	//in %
   PO3_keine_Fkt : INT ;
  END_STRUCT ;
  Datenuebertragung : STRUCT
   Schritt_aktiv : BOOL ;
  END_STRUCT ;
END_VAR
VAR_TEMP
  IO_Adr_Parameterkanal : WORD ;
  IO_Adr_Prozessdatenkanal : WORD ;
  Ret_Val_SFC14_1 : INT ;
  Ret_Val_SFC14_2 : INT ;
  Ret_Val_SFC15_1 : INT ;
  Ret_Val_SFC15_2 : INT ;
  Solldrehzahl_tmp : REAL ;
END_VAR
BEGIN
NETWORK
TITLE = Bausteinende wenn PEA-Adresse = 0
      L     #in_PEA_Adresse;
      L     0;
      ==I;
      BEC;
NETWORK
TITLE = Simulation
//Über die Simulaitonsmerker "M 0.5 Simulation intern" oder "M 0.6 Simulation 
//AVP" 
//wird die Funktion des FUs simuliert:
//- Fehler werden zurückgesetzt
//- Bei Freigabe Istdrehzahl=Solldrehzahl, Betrieb und Solldrehzahl erreicht = 
//True
      O     "M 0.5 InternalSimulation";
      O     "M 0.6 Simulation AVP";
      JCN   NSIM;
      SET;
      R     #out_Stoerung;
      L     L#0;
      T     #out_Stoerungsnummer;
      A     #in_Freigabe;
      =     #out_laeuft;
      =     #out_Sollwert_erreicht;	// (007)
      L     #in_Sollfrequenz;
      JC    SIMD;
      L     0.000000e+00;
SIMD: T     #out_Istfrequenz;
      BEU;
NSIM: NOP   0;
NETWORK
TITLE = Daten von FU einlesen
//UFP-Parameter und FU-Daten auslesen mit SFC14
//PEA_Adresse zeigt auf den Anfang des EA-Bereiches.
// 8-Byte Parameterkanal
      L     #in_PEA_Adresse;
      T     #IO_Adr_Parameterkanal;
      CALL  "SFC 14 DPRD_DAT" (
           LADDR                    := #IO_Adr_Parameterkanal,
           RET_VAL                  := #Ret_Val_SFC14_1,
           RECORD                   := #Parameterkanal_in);
// 6-Byte Prozessdatenkanal
      L     #in_FU_Nummer;
      +     -1;
      L     6;	// Länge eines Parameterkanals je FU
      *I;
      L     #in_PEA_Adresse;
      +I;
      L     8;	// Offset für Parameterkanal
      +I;
      T     #IO_Adr_Prozessdatenkanal;	// Daten des jeweiligen FU = PEA-Adresse + 8 Byte + (FU-Nr. - 1) * 6
      CALL  "SFC 14 DPRD_DAT" (
           LADDR                    := #IO_Adr_Prozessdatenkanal,
           RET_VAL                  := #Ret_Val_SFC14_2,
           RECORD                   := #Prozessdatenkanal_in);
NETWORK
TITLE = Betriebsmeldung
      A     #Prozessdatenkanal_in.PI1_Statuswort.Endstufe_freigegeben;
      A     #Prozessdatenkanal_in.PI1_Statuswort.Umrichter_betriebsbereit;
      A     #Prozessdatenkanal_in.PI1_Statuswort.PA_Daten_freigegeben;
      A(;	// (002)
      L     #Ret_Val_SFC14_2;	// (002)
      L     0;	// (002)
      ==I;	// (002)
      );	// (002)
      =     #out_laeuft;
NETWORK
TITLE = Sollwert erreicht
      L     #in_Sollfrequenz;
      L     #out_Istfrequenz;
      -R;
      ABS;
      L     1.000000e+00;
      <R;
      =     #out_Sollwert_erreicht;
NETWORK
TITLE = Istdrehzahl auswerten
//Istdrehzahl in 0,2 U/min
      L     #Prozessdatenkanal_in.PI2_Istdrehzahl;
      ITD;
      DTR;
      L     5.000000e+00;
      /R;
      T     #out_Istdrehzahl;
NETWORK
TITLE = Istfrequenz auswerten
//Istfrequenz (in Hz) = Istdrehzahl (in 0,2 U/min) / 5 * Nennfrequenz / 
//Nenndrehzahl 
      L     #Prozessdatenkanal_in.PI2_Istdrehzahl;	// (1 == 0,2 U/min)
      ITD;
      DTR;
      L     5.000000e+00;
      /R;
      L     #in_Motornennfrequenz;
      *R;
      L     #in_Motornenndrehzahl;
      /R;
      T     #out_Istfrequenz;	// in Hz
      L     0.000000e+00;	//  wenn kleiner 0 dann negieren 
      <R;
      JCN   E_IF;
      L     #out_Istfrequenz;
      L     -1.000000e+00;
      *R;
      T     #out_Istfrequenz;
E_IF: NOP   0;
NETWORK
TITLE = Stromwert auswerten
      L     #Prozessdatenkanal_in.PI3_Ausgangsstrom;	// in % des FU-Nennstomes 
      ITD;
      DTR;
      L     1.000000e+02;	// (001)
      /R;	// (001)
      L     #in_Motornennstrom;	// (001)
      *R;	// (001)
      T     #out_Ausgangsstrom;
NETWORK
TITLE = Störungsbit auswerten
//Störungsbit aus Statuswort auswerten
//      UN    #Prozessdatenkanal_in.PI1_Statuswort.Umrichter_betriebsbereit    // (004)
      A     #Prozessdatenkanal_in.PI1_Statuswort.Stoerung_Warnung;
      =     #out_Stoerung;
NETWORK
TITLE = Störung resetten
//Störung resetten
      A     #in_Quittierung_Stoerung;
      A     #Prozessdatenkanal_in.PI1_Statuswort.Stoerung_Warnung;
      =     #Prozessdatenkanal_out.PO1_Steuerwort.Reset_Stoerung;
NETWORK
TITLE = Gerätezustand / Störungsnummer des Frequenzumformers auslesen
//Gerätezustand wenn Bit Störung/Warnung = 0
//Störungsnummer wenn Bit Störung/Warnung = 1
      L     #Prozessdatenkanal_in.PI1_Statuswort.Zustand_Fehlercode;
      ITD;
      T     #out_Stoerungsnummer;
// Störmeldung nur wenn Bit Störung = 1
      A     #Prozessdatenkanal_in.PI1_Statuswort.Stoerung_Warnung;
      JC    ESTO;
      L     0;
      T     #out_Stoerungsnummer;
ESTO: NOP   0;
NETWORK
TITLE = Freigabebefehl bearbeiten
//      CLR   // (006)
      AN    #in_Freigabe;	// (006)
      A     #in_Auswahl_Param_satz_2;	// (006)
      AN    #Prozessdatenkanal_in.PI1_Statuswort.akt_Parametersatz_2;	// (006)
      O;
      AN    #in_Freigabe;	// (006)
      AN    #in_Auswahl_Param_satz_2;	// (006)
      A     #Prozessdatenkanal_in.PI1_Statuswort.akt_Parametersatz_2;	// (006)
      =     #Prozessdatenkanal_out.PO1_Steuerwort.Reglersperre;
      SET;
      =     #Prozessdatenkanal_out.PO1_Steuerwort.Freigabe_Schnellstop;
      A     #in_Freigabe;
      =     #Prozessdatenkanal_out.PO1_Steuerwort.Freigabe_Normalhalt;
NETWORK
TITLE = Parametersatz 2 auswählen
//(005) 
//Über dieses Bit kann der Motorparametersatz 2 des FUs angewählt werden
      A     #in_Auswahl_Param_satz_2;	// (005)
      =     #Prozessdatenkanal_out.PO1_Steuerwort.Parametersatz_2;	// (005)
NETWORK
TITLE = Parametersatz 2 auswählen
//(005) 
//Über dieses Bit kann zwischen Integrator 1 und Integrator 2 umgeschaltet werden
//wird nicht verwendet und dauerhaft auf 0 gesetzt
      CLR;	// (005)
      =     #Prozessdatenkanal_out.PO1_Steuerwort.Integratorauswahl;	// (005)
NETWORK
TITLE = Belegung der restlichen Steuerbits
      CLR;
      =     #Prozessdatenkanal_out.PO1_Steuerwort.reserve_3;
      =     #Prozessdatenkanal_out.PO1_Steuerwort.Integratorauswahl;
//      =     #Prozessdatenkanal_out.PO1_Steuerwort.Parametersatz_2 // (005)
      =     #Prozessdatenkanal_out.PO1_Steuerwort.reserve_7;
      =     #Prozessdatenkanal_out.PO1_Steuerwort.Motorpoti_auf;
      =     #Prozessdatenkanal_out.PO1_Steuerwort.Motorpoti_ab;
      =     #Prozessdatenkanal_out.PO1_Steuerwort.Festsollwerte_0;
      =     #Prozessdatenkanal_out.PO1_Steuerwort.Festsollwerte_1;
      =     #Prozessdatenkanal_out.PO1_Steuerwort.Festsollwert_Umschaltung;
      =     #Prozessdatenkanal_out.PO1_Steuerwort.reserve_14;
      =     #Prozessdatenkanal_out.PO1_Steuerwort.reserve_15;
NETWORK
TITLE = Solldrehzahl
//Solldrehzahl (in 0,2 HZ) 
//== Sollfrequenz (in Hz) * 5 * Nenndrehzahl / Nennfrequenz
//
      L     #in_Sollfrequenz;
      L     #in_Motornenndrehzahl;
      *R;
      L     5.000000e+00;
      *R;
      L     #in_Motornennfrequenz;
      /R;
      T     #Solldrehzahl_tmp;	// (003)
      L     3.276700e+04;	// (003)
      >R;	// (003)
      JCN   SD_1;	// (003)
// maximale Drehzahl ausgeben wenn angeforderte größer als Maximalwert ist
      L     3.276700e+04;	// (003)
      RND;	// (003)
      T     #Prozessdatenkanal_out.PO2_Solldrehzahl;	// (003)
      JU    SD_L;	// (003)
// Drehzahl ausgeben wenn angeforderte kleiner als Maximalwert ist
SD_1: L     #Solldrehzahl_tmp;	// (003)
      RND;
      T     #Prozessdatenkanal_out.PO2_Solldrehzahl;
SD_L: AN    #in_Linkslauf;
      JC    E_SD;
      L     #Prozessdatenkanal_out.PO2_Solldrehzahl;
      L     -1;
      *I;
      T     #Prozessdatenkanal_out.PO2_Solldrehzahl;
E_SD: NOP   0;
NETWORK
TITLE = Warnungsbit
//(006) Netzwerk verschoben
//      U     #Prozessdatenkanal_in.PI1_Statuswort.Umrichter_betriebsbereit    // (004)
//      U     #Prozessdatenkanal_in.PI1_Statuswort.Stoerung_Warnung            // (004)
//      O                                        // (004)
      O(;	// (007)
      L     #Solldrehzahl_tmp;	// (006) #Prozessdatenkanal_out.PO2_Solldrehzahl    // (003)
      L     3.276700e+04;	// (003)
      >=R;	// (007)
      );	// (007)
      O(;	// (007)
      L     #Solldrehzahl_tmp;	// (006) #Prozessdatenkanal_out.PO2_Solldrehzahl    // (003)
      L     -3.276700e+04;	// (003)
      <=R;	// (007)
      );	// (007)
      =     #out_Warnung;
NETWORK
TITLE = Netzwerk für nicht unterstützte Funktionen
//Zur Standardisierung der E/A-Parameter aller FUs
      L     0.000000e+00;
      T     #out_Leistung;
      T     #out_Drehmoment;
      T     #out_Motorspannung;
NETWORK
TITLE = Daten an FU senden
// 8-Byte Parameterkanal
      CALL  "SFC 15 DPWR_DAT" (
           LADDR                    := #IO_Adr_Parameterkanal,
           RECORD                   := #Parameterkanal_out,
           RET_VAL                  := #Ret_Val_SFC15_1);
// 6-Byte Prozessdatenkanal
      CALL  "SFC 15 DPWR_DAT" (
           LADDR                    := #IO_Adr_Prozessdatenkanal,
           RECORD                   := #Prozessdatenkanal_out,
           RET_VAL                  := #Ret_Val_SFC15_2);
NETWORK
TITLE = Fehlercode L2Dp in FB_Fehlermeldung
      L     0;
      L     #Ret_Val_SFC14_1;
      <>I;
      JC    Fehl;
      L     0;
      L     #Ret_Val_SFC14_2;
      <>I;
      JC    Fehl;
      L     0;
      L     #Ret_Val_SFC15_1;
      <>I;
      JC    Fehl;
      L     0;
      L     #Ret_Val_SFC15_2;
      <>I;
      JC    Fehl;
      L     0;
Fehl: T     #out_FB_Fehlermeldung;
END_FUNCTION_BLOCK

FUNCTION_BLOCK "FB30 Daten from/to SCADA"	// FB 30
TITLE = copy data from / to SCADA
//Creation:
//Date:            Author:                                               Version
//--------------------------------------------------------------------------------
//14.04.2017      Ilia Bedniakov (ilia)                                  01.00.00
//
//Changes:
//No. Date:        Who       Description                           Mark   Version 
//--------------------------------------------------------------------------------
//01
//________________________________________________________________________________
//Function:
AUTHOR : sra
FAMILY : hsh
VERSION : 0.0
VAR
  reserve_IO : ARRAY  [0 .. 19 ] OF BYTE ;
  date_and_time_CPU : STRUCT
   from_SCADA : STRUCT
    set_actual_date_time : BOOL ;
    set_date_and_time : STRUCT
     year : BYTE ;
     month : BYTE ;
     day : BYTE ;
     hour : BYTE ;
     minoute : BYTE ;
     second : BYTE ;
     milliseconds_h_d : BYTE ;	//milliseconds hundreth and deci position
     milliseconds_u_day : BYTE ;	//milliseconds unit position and day of week (1=Sunday)
    END_STRUCT ;
   END_STRUCT ;
   to_SCADA : STRUCT
    act_date_and_time : STRUCT
     year : BYTE ;
     month : BYTE ;
     day : BYTE ;
     hour : BYTE ;
     minute : BYTE ;
     second : BYTE ;
     milliseconds_h_d : BYTE ;	//milliseconds hundreth and deci position
     milliseconds_u_day : BYTE ;	//milliseconds unit position and day of week (1=Sunday)
    END_STRUCT ;
   END_STRUCT ;
   reserve : ARRAY  [18 .. 19 ] OF BYTE ;
  END_STRUCT ;
  watchdog : STRUCT
   Visualization : ARRAY  [1 .. 10 ] OF STRUCT
    from : INT ;
    to : INT ;
   END_STRUCT ;
   reserve_Watchdog : ARRAY  [40 .. 49 ] OF BYTE ;
  END_STRUCT ;
  fault_messages : STRUCT
   control_bits : STRUCT
    ACK_collective_fault : BOOL ;
    reserve_0_1 : BOOL ;
    reserve_0_2 : BOOL ;
    reserve_0_3 : BOOL ;
    reserve_0_4 : BOOL ;
    reserve_0_5 : BOOL ;
    reserve_0_6 : BOOL ;
    reserve_0_7 : BOOL ;
   END_STRUCT ;
   status_bits : STRUCT
    collective_fault : BOOL ;
    fault_fuse : BOOL ;
    reserve_0_2 : BOOL ;
    reserve_0_3 : BOOL ;
    reserve_0_4 : BOOL ;
    reserve_0_5 : BOOL ;
    reserve_0_6 : BOOL ;
    reserve_0_7 : BOOL ;
   END_STRUCT ;
   reserve : ARRAY  [4 .. 9 ] OF BYTE ;
  END_STRUCT ;
  system_on_off : STRUCT
   system_area : ARRAY  [1 .. 10 ] OF STRUCT
    control_bits : STRUCT
     system_on : BOOL ;
     system_off : BOOL ;
     reserve_0_2 : BOOL ;
     reserve_0_3 : BOOL ;
     reserve_0_4 : BOOL ;
     reserve_0_5 : BOOL ;
     reserve_0_6 : BOOL ;
     reserve_0_7 : BOOL ;
    END_STRUCT ;
    status_bits : STRUCT
     system_on : BOOL ;	//1= System on
     emergency_stop : BOOL ;	//1= Emergency stop OK (0= display = blue)
     reserve_0_2 : BOOL ;
     reserve_0_3 : BOOL ;
     reserve_0_4 : BOOL ;
     reserve_0_5 : BOOL ;
     reserve_0_6 : BOOL ;
     reserve_0_7 : BOOL ;
    END_STRUCT ;
   END_STRUCT ;
   reserve : ARRAY  [40 .. 99 ] OF BYTE ;
  END_STRUCT ;
  mode_switches : STRUCT
   from_SCADA : STRUCT
    service_mode_released : BOOL ;	//TRUE = service mode released
    Second_service_mode : BOOL ;	//TRUE = service mode available during auto run
    light_test : BOOL ;	//TRUE = light test
    automatic_mode_line : ARRAY  [1 .. 64 ] OF //FALSE = auto mode; TRUE = manual mode
    BOOL ;
    reserve : ARRAY  [10 .. 19 ] OF BYTE ;
   END_STRUCT ;
   to_SCADA : STRUCT
    RLS_service_mode_on : BOOL ;	//TRUE = release service mode switch for motor and valve objects
    RLS_second_service_mode : BOOL ;	//TRUE = release service mode switch for motor and valve objects
    RLS_manual_to_auto_line : ARRAY  [1 .. 64 ] OF //TRUE = release for mode switch of line, area, mixer from manual to auto
    BOOL ;
    RLS_auto_to_manual_line : ARRAY  [1 .. 64 ] OF //TRUE = release for mode switch of line, area, mixer from auto to manual
    BOOL ;
    reason_switch_locked : STRUCT 	//explanation why mode switch is locked (option)
     service_mode : INT ;
     manual_auto_line : ARRAY  [1 .. 64 ] OF INT ;
    END_STRUCT ;
   END_STRUCT ;
   reserve : ARRAY  [168 .. 199 ] OF BYTE ;
  END_STRUCT ;
  reserve : ARRAY  [400 .. 499 ] OF BYTE ;
  BatchInfo : STRUCT
   Line1 : STRUCT
    SC11 : STRUCT
     order_number : ARRAY  [0 .. 19 ] OF CHAR ;
     batch_number : INT ;
     reserve : ARRAY  [22 .. 49 ] OF BYTE ;
    END_STRUCT ;
    FH11 : STRUCT
     order_number : ARRAY  [0 .. 19 ] OF CHAR ;
     batch_number : INT ;
     reserve : ARRAY  [22 .. 49 ] OF BYTE ;
    END_STRUCT ;
    BH11 : STRUCT
     order_number : ARRAY  [0 .. 19 ] OF CHAR ;
     batch_number : INT ;
     reserve : ARRAY  [22 .. 49 ] OF BYTE ;
    END_STRUCT ;
   END_STRUCT ;
   Line2 : STRUCT
    SC21 : STRUCT
     order_number : ARRAY  [0 .. 19 ] OF CHAR ;
     batch_number : INT ;
     reserve : ARRAY  [22 .. 49 ] OF BYTE ;
    END_STRUCT ;
    FH21 : STRUCT
     order_number : ARRAY  [0 .. 19 ] OF CHAR ;
     batch_number : INT ;
     reserve : ARRAY  [22 .. 49 ] OF BYTE ;
    END_STRUCT ;
    BH21 : STRUCT
     order_number : ARRAY  [0 .. 19 ] OF CHAR ;
     batch_number : INT ;
     reserve : ARRAY  [22 .. 49 ] OF BYTE ;
    END_STRUCT ;
   END_STRUCT ;
   Line3 : STRUCT
    SC31 : STRUCT
     order_number : ARRAY  [0 .. 19 ] OF CHAR ;
     batch_number : INT ;
     reserve : ARRAY  [22 .. 49 ] OF BYTE ;
    END_STRUCT ;
    FH31 : STRUCT
     order_number : ARRAY  [0 .. 19 ] OF CHAR ;
     batch_number : INT ;
     reserve : ARRAY  [22 .. 49 ] OF BYTE ;
    END_STRUCT ;
    BH31 : STRUCT
     order_number : ARRAY  [0 .. 19 ] OF CHAR ;
     batch_number : INT ;
     reserve : ARRAY  [22 .. 49 ] OF BYTE ;
    END_STRUCT ;
   END_STRUCT ;
  END_STRUCT ;
  INTERNAL : STRUCT
   Flags : STRUCT
    reserve : BOOL ;
    reserve_1 : BOOL ;
    reserve_2 : BOOL ;
    reserve_3 : BOOL ;
    reserve_4 : BOOL ;
    reserve_5 : BOOL ;
    reserve_6 : BOOL ;
    reserve_7 : BOOL ;
    reserve_8 : BOOL ;
    reserve_9 : BOOL ;
    reserve_10 : BOOL ;
    reserve_11 : BOOL ;
    reserve_12 : BOOL ;
    reserve_13 : BOOL ;
    reserve_14 : BOOL ;
    reserve_15 : BOOL ;
   END_STRUCT ;
  END_STRUCT ;
END_VAR
VAR_TEMP
  set_date_and_time : DATE_AND_TIME ;
  act_date_and_time : DATE_AND_TIME ;
  Ret_Val_SFC0_SFC1 : INT ;
  copyerror : INT ;
END_VAR
BEGIN
NETWORK
TITLE = set date and time
//transformation from integer to BCD
      A     DB30.DBX 20.0;
//      SET   
      =     DB30.DBX 20.0;
      AN    #date_and_time_CPU.from_SCADA.set_actual_date_time;
      JC    E_DT;
      LAR1  P##set_date_and_time;
      L     #date_and_time_CPU.from_SCADA.set_date_and_time.year;
//      ITB   
      T     LB [AR1,P#0.0];
      L     #date_and_time_CPU.from_SCADA.set_date_and_time.month;
//      ITB   
      T     LB [AR1,P#1.0];
      L     #date_and_time_CPU.from_SCADA.set_date_and_time.day;
//      ITB   
      T     LB [AR1,P#2.0];
      L     #date_and_time_CPU.from_SCADA.set_date_and_time.hour;
//      ITB   
      T     LB [AR1,P#3.0];
      L     #date_and_time_CPU.from_SCADA.set_date_and_time.minoute;
//      ITB   
      T     LB [AR1,P#4.0];
      L     #date_and_time_CPU.from_SCADA.set_date_and_time.second;
//      ITB   
      T     LB [AR1,P#5.0];
      L     #date_and_time_CPU.from_SCADA.set_date_and_time.milliseconds_h_d;
//      ITB   
      T     LB [AR1,P#6.0];
      L     #date_and_time_CPU.from_SCADA.set_date_and_time.milliseconds_u_day;
//      ITB   
      T     LB [AR1,P#7.0];
      CALL  "SET_CLK" (
           PDT                      := #set_date_and_time,
           RET_VAL                  := #Ret_Val_SFC0_SFC1);
      SET;
      R     #date_and_time_CPU.from_SCADA.set_actual_date_time;
E_DT: NOP   0;
NETWORK
TITLE = read date and time
      CALL  "READ_CLK" (
           RET_VAL                  := #Ret_Val_SFC0_SFC1,
           CDT                      := #act_date_and_time);
NETWORK
TITLE = actual date and time transformation
//transformation from BCD to integer
      LAR1  P##act_date_and_time;
      L     LB [AR1,P#0.0];
//      BTI   
      T     #date_and_time_CPU.to_SCADA.act_date_and_time.year;
      L     LB [AR1,P#1.0];
//      BTI   
      T     #date_and_time_CPU.to_SCADA.act_date_and_time.month;
      L     LB [AR1,P#2.0];
//      BTI   
      T     #date_and_time_CPU.to_SCADA.act_date_and_time.day;
      L     LB [AR1,P#3.0];
//      BTI   
      T     #date_and_time_CPU.to_SCADA.act_date_and_time.hour;
      L     LB [AR1,P#4.0];
//      BTI   
      T     #date_and_time_CPU.to_SCADA.act_date_and_time.minute;
      L     LB [AR1,P#5.0];
//      BTI   
      T     #date_and_time_CPU.to_SCADA.act_date_and_time.second;
      L     LB [AR1,P#6.0];
//      BTI   
      T     #date_and_time_CPU.to_SCADA.act_date_and_time.milliseconds_h_d;
      L     LB [AR1,P#7.0];
//      BTI   
      T     #date_and_time_CPU.to_SCADA.act_date_and_time.milliseconds_u_day;
NETWORK
TITLE = collective fault and acknowledgement
      A     #fault_messages.control_bits.ACK_collective_fault;
      =     "M 1.0 Ack. faults";
      A     "M 1.1 general Fault";
      =     #fault_messages.status_bits.collective_fault;
NETWORK
TITLE = Service Mode (Motor + Ventile)
//Service Mode zentral sperren
      AN    #mode_switches.from_SCADA.service_mode_released;
      =     "M 0.0 Lock Man.Operation";
      SET;
      =     #mode_switches.to_SCADA.RLS_service_mode_on;
//Freigabe für Service Mode Schalter aus SPS
//      SET   
//      =     #mode_switches.to_SCADA.RLS_second_service_mode
// Das brauchen wir nicht!!!!!!
//second service mode
//      A     #mode_switches.from_SCADA.Second_service_mode
//      =     "Service mode lock auto"
//release switch second service mode
//      SET   
//      =     #mode_switches.to_SCADA.RLS_second_service_mode
NETWORK
TITLE = system on
      A     #system_on_off.system_area[1].control_bits.system_on;
      A     "ES_03_01_601";
      S     #system_on_off.system_area[1].status_bits.system_on;
      O     #system_on_off.system_area[1].control_bits.system_off;
      ON    "ES_03_01_601";
      R     #system_on_off.system_area[1].status_bits.system_on;
      A     "ES_03_01_601";
      =     #system_on_off.system_area[1].status_bits.emergency_stop;
      AN    #system_on_off.system_area[1].status_bits.system_on;
      =     DB34.DBX 1000.2;
NETWORK
TITLE = Sys. general Faults to VISU 
// emergency Stop not active
      AN    "ES_03_01_601";
      =     DB34.DBX 5.6;
// fault fuse
      AN    "ES_03_01_602";
      =     #fault_messages.status_bits.fault_fuse;
      =     DB34.DBX 5.7;
END_FUNCTION_BLOCK

FUNCTION_BLOCK "FB32 Inputs to SCADA"	// FB 32
TITLE = Inputs for SCADA
AUTHOR : sra
FAMILY : SCADA
NAME : inputs
VERSION : 0.0
VAR
  input : ARRAY  [0 .. 1023, 0 .. 7 ] OF BOOL ;
END_VAR
VAR_TEMP
  Fault_Block_copy : INT ;
END_VAR
BEGIN
NETWORK
TITLE = Copy Image of Inputs for SCADA in DB32
      CALL  "FC5 Block Transfer" (
           Quell_Typ                := B#16#45,
           Quell_DB                 := 0,
           Quell_DW                 := 0,
           Ziel_Typ                 := B#16#49,
           Ziel_DB                  := 32,
           Ziel_DW                  := 0,
           Block_Laenge             := 128,
           outFehler                := #Fault_Block_copy);
END_FUNCTION_BLOCK

FUNCTION_BLOCK "FB33 Outputs to SCADA"	// FB 33
TITLE = Outputs for SCADA
AUTHOR : sra
FAMILY : SCADA
NAME : outputs
VERSION : 0.0
VAR
  output : ARRAY  [0 .. 1023, 0 .. 7 ] OF BOOL ;
END_VAR
VAR_TEMP
  Fault_Block_copy : INT ;
END_VAR
BEGIN
NETWORK
TITLE = Copy Image of Outputs for SCADA in DB33
      CALL  "FC5 Block Transfer" (
           Quell_Typ                := B#16#41,
           Quell_DB                 := 0,
           Quell_DW                 := 0,
           Ziel_Typ                 := B#16#49,
           Ziel_DB                  := 33,
           Ziel_DW                  := 0,
           Block_Laenge             := 128,
           outFehler                := #Fault_Block_copy);
END_FUNCTION_BLOCK

FUNCTION_BLOCK "FB34 Fault evaluation"	// FB 34
TITLE = Fault evaluation
//Building:
//Date         Editor                                                     Version
//--------------------------------------------------------------------------------
//
//
//Modifications:
//No. Date     Edit  Description                                    Index Version
//--------------------------------------------------------------------------------
// 
AUTHOR : sra
FAMILY : AZO
VERSION : 0.0
VAR
  Stoerung_E : ARRAY  [0 .. 1023, 0 .. 7 ] OF BOOL ;
  Erstwertmeldung_E : ARRAY  [0 .. 1023, 0 .. 7 ] OF BOOL ;
  Spiegelung_PC_Fehler_E : ARRAY  [0 .. 1023, 0 .. 7 ] OF BOOL ;
  Quittierung_von_PC_E : ARRAY  [0 .. 1023, 0 .. 7 ] OF BOOL ;
  Quittierung_von_OP : ARRAY  [0 .. 1023, 0 .. 7 ] OF //acknowledge bits from Siemens panel
  BOOL ;
  alte_Quittieung_von_OP : ARRAY  [0 .. 1023, 0 .. 7 ] OF //acknowledge bits from Siemens panel one cycle before
  BOOL ;
END_VAR
VAR_TEMP
  Ack_Fault : BOOL ;
END_VAR
BEGIN
NETWORK
TITLE = CPU Fehler
      L     DB3.DBW 30;
      T     DB34.DBW 0;
NETWORK
TITLE = Quit faults
      A     "M 1.0 Ack. faults";
      =     #Ack_Fault;
NETWORK
TITLE = Erstwertmeldung / Quittierung
      CALL  "FC16 Fault evaluation" (
           Conf_AckBySiemensOP      := TRUE,
           Stoerungstakt            := "M 4.7 Imp Cycle 2,0-sec",
           Freigabe_Sammelstoerung  := TRUE,
           Quittierung              := #Ack_Fault,
           Stoerungs_DB             := 34,
           Quittierungs_DB_SCADA    := 35,
           Anzahl_Stoerungs_Byte    := 1024,
           Offset_Stoerungs_Byte    := 0,
           Adresse_Anfangswort      := 0,
           Bereichslaenge           := 1024,
           Sammelstoerung           := "M 1.1 general Fault",
           Erstmeldung              := "M 1.2 First-out Fault",
           Erstmeldung_PC           := "M 8.0 First-out alarm PC",
           Quittierung_PC           := "M 8.1 ACK Fault from PC");	// FALSE   //wenn OP vorhanden ist muss dasd Bit gesetzt werden
NETWORK
TITLE = collective fault / horn
//e.g. customer can connect a lamp
      A     "M 1.1 general Fault";
      A     "M 1.2 First-out Fault";
      A     "M 2.5 Cycle 1,0-sec";
      O;
      A     "M 1.1 general Fault";
      AN    "M 1.2 First-out Fault";
      =     "ES_02_03_505";
NETWORK
TITLE = CPU Fehler löschen
      L     DB3.DBW 30;
      L     DB35.DBW 0;
      INVI;
      AW;
      T     DB3.DBW 30;
END_FUNCTION_BLOCK

FUNCTION_BLOCK "PRODUCTION"	// FB 1000
TITLE = Call Production FB's
//Creation:
//Date:            Author:                                               Version
//--------------------------------------------------------------------------------
//14.04.2017      Ilia Bedniakov(ilia)                                   01.00.00
//
//Changes:
//No. Date:        Who       Description                           Mark   Version 
//--------------------------------------------------------------------------------
//01
//________________________________________________________________________________
//Function:
VERSION : 0.1
VAR_TEMP
  dummy_bool : BOOL ;
END_VAR
BEGIN
NETWORK
TITLE = Call Receiver REC01 FB
      CALL  "REC01" , "REC01_DB" (
           IF_Blower_DB             := 1051,
           IF_Blower_DW             := 200,
           iSystemActive            := DB30.DBX 102.0,
           iSafetySwitchRF_ok       := "GZ_02_01_601",
           iToolKeyControlRF_ok     := "Gn_02_01_602",
           iSafetySwitchMS_ok       := "GZ_02_02_601",
           iPFCPM_Ready             := "ES_02_03_601",
           iPFCPM_TakeProduct       := "ES_02_03_602",
           iRepRotaryFeeder_on      := "HZ_02_01_201",
           iRepScreener_on          := "HZ_02_02_201",
           iRepMetalSeparator_on    := "HZ_02_02_202",
           iFBRotaryFeeder_on       := "EUi_02_01_201",
           iFBScreener_on           := "EUi_02_02_201",
           iFBMetalSeparator_on     := "EUi_02_02_202",
           iHighLevelREC01_free     := "Lp_02_01_301",
           iLowLevelREC01_free      := "Ln_02_01_302",
           iHighLevelHP03_free      := "Lp_02_03_301",
           iLowLevelHP03_free       := "Ln_02_03_302",
           aRepRotaryValve          := "DB35 Acknowledge Faults".Quittierung[5, 1],
           aRepScreener             := "DB35 Acknowledge Faults".Quittierung[5, 2],
           aRepMetalSeparator       := "DB35 Acknowledge Faults".Quittierung[5, 3],
           aFBRotaryValve           := "DB35 Acknowledge Faults".Quittierung[4, 1],
           aFBScreener              := "DB35 Acknowledge Faults".Quittierung[4, 2],
           aFBMetalSeparator        := "DB35 Acknowledge Faults".Quittierung[4, 3],
           aSafetySwitchRV          := "DB35 Acknowledge Faults".Quittierung[6, 0],
           aToolKeyControlRF        := "DB35 Acknowledge Faults".Quittierung[6, 4],
           aSafetySwitchSM          := "DB35 Acknowledge Faults".Quittierung[6, 1],
           aFullREC01               := "DB35 Acknowledge Faults".Quittierung[10, 0],
           aSiloNrNotCorrect        := "DB35 Acknowledge Faults".Quittierung[1001, 1],
           qRotaryValve_on          := "EUq_02_01_201",
           qScreener_on             := "EUq_02_02_201",
           qMetalSeparator_on       := "EUq_02_02_202",
           qAPBRotaryValve_on       := "UVp_02_01_101",
           qPurgingFilterV1_on      := "UVp_02_01_102",
           qPurgingFilterV2_on      := "UVp_02_01_103",
           qPurgingFilterV3_on      := "UVp_02_01_104",
           qPFCPM_Product           := "ES_02_03_501",
           qPFCPM_Active            := "ES_02_03_502",
           fRepRotaryValve          := DB34.DBX 5.1,
           fRepScreener             := DB34.DBX 5.2,
           fRepMetalSeparator       := DB34.DBX 5.3,
           fFBRotaryFeeder          := DB34.DBX 4.1,
           fFBScreener              := DB34.DBX 4.2,
           fFBMetalSeparator        := DB34.DBX 4.3,
           fSafetyRotaryFeeder      := DB34.DBX 6.0,
           fToolKeyControl          := DB34.DBX 6.4,
           fSafetyMS                := DB34.DBX 6.1,
           fREC01HighLevel          := DB34.DBX 10.0,
           fHP03HighLevel           := DB34.DBX 10.2,
           fREC01_LLCovered         := DB34.DBX 10.1,
           fSiloNrNotCorrect        := DB34.DBX 1001.1,
           fLineNotEmpty            := DB34.DBX 1001.2);	// ak
NETWORK
TITLE = Call Blower FB1051
      CALL  "PMP01" , "PMP01_DB" (
           piwPressure              := 128,
           SystemActive             := DB30.DBX 102.0,
           iFBBlower_on             := "EUi_02_04_201",
           iRepBlower_on            := "HZ_02_04_201",
           aFBBlower                := "DB35 Acknowledge Faults".Quittierung[4, 0],
           aRepBlower               := "DB35 Acknowledge Faults".Quittierung[5, 0],
           qBlower_on               := "EUq_02_04_201",
           fFBBlower                := DB34.DBX 4.0,
           fRepBlower               := DB34.DBX 5.0,
           fPressureFault           := DB34.DBX 1002.0,
           wBrokenWirePT            := DB34.DBX 1002.1);
NETWORK
TITLE = Call HP01
      CALL  "HOPPER" , "HOPPER_HP01_DB" (
           in_HopperNumber          := 1,
           IF_FC_RotaryFeeder_DB    := 10001,
           IF_FC_RotaryFeeder_DW    := 100,
           SystemActive             := DB30.DBX 102.0,
           iLowLevelHopper          := "Ln_01_01_301",
           iRepRotaryFeeder         := "HZ_01_01_201",
           iRepVibrator1            := "HZ_01_01_202",
           iRepVibrator2            := #dummy_bool,
           iFBVibrator1_on          := "EUi_01_01_202",
           iFBVibrator2_on          := #dummy_bool,
           iFBRotaryFeeder_on       := "EUi_01_01_201",
           iProductValve_open       := TRUE,
           iSafetyRotaryFeeder_ok   := "GZ_01_01_601",
           iSafetyToolKeyControl    := "Gn_01_01_602",
           aFBRotaryFeeder          := "DB35 Acknowledge Faults".Quittierung[4, 4],
           aFBVibrator1             := "DB35 Acknowledge Faults".Quittierung[10, 5],
           aFBVibrator2             := #dummy_bool,
           aRepRotaryValve          := "DB35 Acknowledge Faults".Quittierung[5, 4],
           aRepVibrator1            := "DB35 Acknowledge Faults".Quittierung[11, 0],
           aRepVibrator2            := #dummy_bool,
           aSafetyRotaryFeeder      := "DB35 Acknowledge Faults".Quittierung[6, 2],
           aToolKeyControl          := "DB35 Acknowledge Faults".Quittierung[6, 5],
           qRotaryFeeder_on         := "EUq_01_01_201",
           qAPBRotaryFeeder         := "UVp_01_01_101",
           qVibrator1               := "EUq_01_01_202",
           qVibrator2               := #dummy_bool,
           fFBRotaryFeeder          := DB34.DBX 4.4,
           fFBVibrator1             := DB34.DBX 10.5,
           fFBVibrator2             := #dummy_bool,
           fRepRotaryFeeder         := DB34.DBX 5.4,
           fRepVibrator1            := DB34.DBX 11.0,
           fRepVibrator2            := #dummy_bool,
           fSafetyRotaryFeeder      := DB34.DBX 6.2,
           fToolKeyControl          := DB34.DBX 6.5,
           fProductFlap             := #dummy_bool);	// "DB35 Acknowledge Faults".Quittierung[10, 5]
NETWORK
TITLE = Call HP02
      CALL  "HOPPER" , "HOPPER_HP02_DB" (
           in_HopperNumber          := 2,
           IF_FC_RotaryFeeder_DB    := 10001,
           IF_FC_RotaryFeeder_DW    := 100,
           SystemActive             := DB30.DBX 102.0,
           iLowLevelHopper          := "Ln_01_02_301",
           iRepRotaryFeeder         := "HZ_01_02_201",
           iRepVibrator1            := "HZ_01_02_202",
           iRepVibrator2            := "HZ_01_02_203",
           iFBVibrator1_on          := "EUi_01_02_202",
           iFBVibrator2_on          := "EUi_01_02_203",
           iFBRotaryFeeder_on       := "EUi_01_02_201",
           iProductValve_open       := "Gp_01_02_102",
           iSafetyRotaryFeeder_ok   := "GZ_01_02_601",
           iSafetyToolKeyControl    := "Gn_01_02_602",
           aFBRotaryFeeder          := "DB35 Acknowledge Faults".Quittierung[4, 5],
           aFBVibrator1             := "DB35 Acknowledge Faults".Quittierung[10, 6],
           aFBVibrator2             := "DB35 Acknowledge Faults".Quittierung[10, 7],
           aRepRotaryValve          := "DB35 Acknowledge Faults".Quittierung[5, 5],
           aRepVibrator1            := "DB35 Acknowledge Faults".Quittierung[11, 1],
           aRepVibrator2            := "DB35 Acknowledge Faults".Quittierung[11, 2],
           aSafetyRotaryFeeder      := "DB35 Acknowledge Faults".Quittierung[6, 3],
           aToolKeyControl          := "DB35 Acknowledge Faults".Quittierung[6, 6],
           qRotaryFeeder_on         := "EUq_01_02_201",
           qAPBRotaryFeeder         := "UVp_01_02_101",
           qVibrator1               := "EUq_01_02_202",
           qVibrator2               := "EUq_01_02_203",
           fFBRotaryFeeder          := DB34.DBX 4.5,
           fFBVibrator1             := DB34.DBX 10.6,
           fFBVibrator2             := DB34.DBX 10.7,
           fRepRotaryFeeder         := DB34.DBX 5.5,
           fRepVibrator1            := DB34.DBX 11.1,
           fRepVibrator2            := DB34.DBX 11.2,
           fSafetyRotaryFeeder      := DB34.DBX 6.3,
           fToolKeyControl          := DB34.DBX 6.6,
           fProductFlap             := DB34.DBX 10.4);
NETWORK
TITLE = Call Frequency Converter
      CALL  "FC01_RV_HOPPERS" , "FC01_RV_HOPPERS_DB" (
           in_FU_Typ                := 6,
           in_PEA_Adresse           := 400,
           in_FU_Nummer             := 1,
           in_Motornennfrequenz     := 5.000000e+01,
           in_Motornenndrehzahl     := 1.435000e+03,
           FU_Stoerung              := DB34.DBX 1000.0);
END_FUNCTION_BLOCK

